FUNCTION FUN_RetractStorageCylinder : BOOL
VAR_INPUT
END_VAR
VAR
END_VAR

END_FUNCTION

(* stored: Version 1.1.0.1, ProductVersion 3.1.4024.13
   POU FUN_RetractStorageCylinder: Id {0b8cab62-7e15-4d8b-8223-49aced03d0ff}, SpecialFunc None *)
